// TIA Portal V20 export
VAR_GLOBAL   // PLC tag table "plant"
   DoorOpenRequest AT %M200.0 : Bool;
END_VAR
